(* CODESYS project tctwinsafe.library
   Title: Tc2_TwinSAFE
   Version: 1.0.0.0
   Placeholder: Tc2_TwinSAFE
   Company: Beckhoff Automation GmbH

Project tree, tasks and I/O mapping:
  libraries: Tc2_System, * (Beckhoff Automation GmbH)
  Data types/
    data type TwinSAFE_Data
  Global Variables/
    global variables Globale_Variablen
  POUs/
    function F_GetVersionTcTwinSAFE [ST]
    function block FB_TwinSAFE_connection [ST]
  Version/
    global variables Global_Version
  Visualizations/
*)

// Data types/TwinSAFE_Data
TYPE TwinSAFE_Data :
ARRAY[0..5] OF BYTE;
END_TYPE

// Global Variables/Globale_Variablen
VAR_GLOBAL
END_VAR

// Version/Global_Version
// This function has been automatically generated from the project information.
VAR_GLOBAL CONSTANT
	{attribute 'const_non_replaced'}
	stLibVersion_Tc2_TwinSAFE : ST_LibVersion := (iMajor := 1, iMinor := 0, iBuild := 0, iRevision := 0, sVersion := '1.0.0.0');
END_VAR

// POUs/F_GetVersionTcTwinSAFE
(*
DATE          | Version    | created under        | Author          | Remark
----------------------------------------------------------------------------------------
01/09/2008    | 0.0.1      | V2.10.0 (Build 1321) | O. Ellerbrock   | start of implementation
02/28/2008    | 1.0.0      | V2.10.0 (Build 1323) | O. Ellerbrock   | Release
*)
FUNCTION F_GetVersionTcTwinSAFE : UINT
VAR_INPUT
       nVersionElement       :       INT;
END_VAR
VAR
END_VAR


CASE nVersionElement OF
1: (* major number *)
       F_GetVersionTcTwinSAFE := 1;
2: (* minor number *)
       F_GetVersionTcTwinSAFE := 0;
3: (* revision number *)
       F_GetVersionTcTwinSAFE := 0;
ELSE
   F_GetVersionTcTwinSAFE := 16#FFFF;
END_CASE

END_FUNCTION

// POUs/FB_TwinSAFE_connection
FUNCTION_BLOCK FB_TwinSAFE_connection
(*
The function block FB_TwinSAFE_connection is made for evaluating the TwinSAFE data which is transfered 
from one TwinSAFE communication partner to another TwinSAFE communication partner. The input 
parameters has to be linked to the SafetyQBx or SafetyIn signal of the corresponding TwinSAFE terminal. 
Please assure that the new linkage does not remove the already existing linkage. When RT Ethernet is used 
to transfer the TwinSAFE data, one parameter has to be linked to SafetyQBx the other parameter has to be linked 
to Vardata of the network variable subscriber. 
*)
VAR_INPUT
	TwinSAFETerminal AT %I* : TwinSAFE_Data; (* Additional link to "SafetyIn" e.g. KL1904, KL2904, network variable subscriber*)
	TwinSAFELogic AT %I* : TwinSAFE_Data; (* Additional link to "SafetyQBx" e.g. KL6904 *)
END_VAR
VAR_OUTPUT
	nSafeTerminalData : BYTE; (* TwinSAFE data of SafetyIn e.g. KL1904, KL2904, network variable subscriber *)
	nSafeLogicData : BYTE; (* TwinSAFE data of SafetyOut *)
	tCycleTime: TIME; (* Cycletime in ms *)
	bConnectionInRun : BOOL; (* Connection in RUN *)
	nFirstError : WORD; (* First error in connection *)
	nLastError : WORD; (* Last error in connection *)
END_VAR


VAR
	TwinSAFE_OldInMessage : TwinSAFE_Data;
	OldInCounter : UDINT;
	bConnectionInInRun : BOOL;
	bConnectionOutInRun : BOOL;
	nErrorIn1 : BYTE;
	nErrorIn11 : BYTE;
	nErrorIn2 : BYTE;
	nErrorOut1 : BYTE;
	nErrorOut11 : BYTE;
	nErrorOut2 : BYTE;
	nLastErrorTemp : WORD; (* Last error in connection *)
	Tasknummer: INT := 1; (* Tasknumber of task in which this FB is executed *)
	GETCURTASKINDEX_1: GETCURTASKINDEX;
END_VAR

(* Get Tasknumber of task in which this FB is executed *)
GETCURTASKINDEX_1();
Tasknummer := GETCURTASKINDEX_1.index;

(* Input TwinSAFETerminal *)
CASE TwinSAFETerminal[0] OF

0: (* TwinSAFE *)
	IF TwinSAFETerminal[2] = 0 AND NOT
		(TwinSAFETerminal[1] = 0 AND TwinSAFETerminal[3] = 0 AND TwinSAFETerminal[4] = 0 AND TwinSAFETerminal[5] = 0) THEN
		nSafeTerminalData := TwinSAFETerminal[1];
		bConnectionInInRun := TRUE;
	ELSE
		nSafeTerminalData := 0;
		bConnectionInInRun := FALSE;
	END_IF
	(* Checking for errors *)
	IF TwinSAFETerminal[2] <> 0 AND NOT
		(TwinSAFETerminal[4] = 0 AND TwinSAFETerminal[5] = 0) THEN
		nErrorIn1 := TwinSAFETerminal[2];
		nErrorIn11 := TwinSAFETerminal[0];
	END_IF

	(* Zeitmessung *)
	IF TwinSAFETerminal[3] <> TwinSAFE_OldInMessage[3] THEN
		tCycleTime := UDINT_TO_TIME(((TwinCAT_SystemInfoVarList._TaskInfo[Tasknummer].CycleCount -
		OldInCounter)*  TwinCAT_SystemInfoVarList._TaskInfo[Tasknummer].CycleTime)/10000);
		IF OldInCounter = 0 THEN
			tCycleTime := t#0ms;
		END_IF
		OldInCounter :=  TwinCAT_SystemInfoVarList._TaskInfo[Tasknummer].CycleCount;
		TwinSAFE_OldInMessage := TwinSAFETerminal;
	END_IF

1: (* TwinSAFE *)
	IF TwinSAFETerminal[2] = 0 AND NOT
		(TwinSAFETerminal[4] = 0 AND TwinSAFETerminal[5] = 0) THEN
		nSafeTerminalData := TwinSAFETerminal[1];
		bConnectionInInRun := TRUE;
	ELSE
		nSafeTerminalData := 0;
		bConnectionInInRun := FALSE;
	END_IF
	(* Checking for errors *)
	IF TwinSAFETerminal[2] <> 0 AND NOT
		(TwinSAFETerminal[4] = 0 AND TwinSAFETerminal[5] = 0) THEN
		nErrorIn1 := TwinSAFETerminal[2];
		nErrorIn11 := TwinSAFETerminal[0];
	END_IF

	(* Zeitmessung *)
	IF TwinSAFETerminal[3] <> TwinSAFE_OldInMessage[3] THEN
		tCycleTime := UDINT_TO_TIME(((TwinCAT_SystemInfoVarList._TaskInfo[Tasknummer].CycleCount -
		OldInCounter)*  TwinCAT_SystemInfoVarList._TaskInfo[Tasknummer].CycleTime)/10000);
		IF OldInCounter = 0 THEN
			tCycleTime := t#0ms;
		END_IF
		OldInCounter :=  TwinCAT_SystemInfoVarList._TaskInfo[Tasknummer].CycleCount;
		TwinSAFE_OldInMessage := TwinSAFETerminal;
	END_IF


16#08, 16#2A, 16#4E, 16#52, 16#64: (* Safety over EtherCAT, FailSafe-Data *)
	nSafeTerminalData := 0;
	bConnectionInInRun := FALSE;
	(* Checking for error *)
	IF TwinSAFETerminal[0] = 16#2A THEN
		nErrorIn2 := TwinSAFETerminal[1];
	END_IF
	(* Zeitmessung *)
	IF (TwinSAFETerminal[2] <> TwinSAFE_OldInMessage[2]) OR
		(TwinSAFETerminal[3] <> TwinSAFE_OldInMessage[3])  THEN
		tCycleTime := UDINT_TO_TIME(((TwinCAT_SystemInfoVarList._TaskInfo[Tasknummer].CycleCount -
		OldInCounter)*  TwinCAT_SystemInfoVarList._TaskInfo[Tasknummer].CycleTime)/10000);
		IF OldInCounter = 0 THEN
			tCycleTime := t#0ms;
		END_IF
		OldInCounter :=  TwinCAT_SystemInfoVarList._TaskInfo[Tasknummer].CycleCount;
		TwinSAFE_OldInMessage := TwinSAFETerminal;
	END_IF

16#36: (* Safety over EtherCAT, Data*)
	nSafeTerminalData := TwinSAFETerminal[1];
	bConnectionInInRun := TRUE;
	(* Zeitmessung *)
	IF (TwinSAFETerminal[2] <> TwinSAFE_OldInMessage[2]) OR
		(TwinSAFETerminal[3] <> TwinSAFE_OldInMessage[3])  THEN
		tCycleTime := UDINT_TO_TIME(((TwinCAT_SystemInfoVarList._TaskInfo[Tasknummer].CycleCount -
		OldInCounter)*  TwinCAT_SystemInfoVarList._TaskInfo[Tasknummer].CycleTime)/10000);
		IF OldInCounter = 0 THEN
			tCycleTime := t#0ms;
		END_IF
		OldInCounter :=  TwinCAT_SystemInfoVarList._TaskInfo[Tasknummer].CycleCount;
		TwinSAFE_OldInMessage := TwinSAFETerminal;
	END_IF

ELSE
(* Inputs auf 0 setzen *)
	nSafeTerminalData := 0;
	tCycleTime := t#0ms;
	bConnectionInInRun := FALSE;
END_CASE



(* Input TwinSAFELogic *)
CASE TwinSAFELogic[0] OF

0: (* TwinSAFE Protokoll *)
	IF TwinSAFELogic[2] = 0 AND NOT
		(TwinSAFELogic[4] = 0 AND TwinSAFELogic[5] = 0) THEN
		nSafeLogicData := TwinSAFELogic[1];
		bConnectionOutInRun := TRUE;
	ELSE
		nSafeLogicData := 0;
		bConnectionOutInRun := FALSE;
	END_IF
	(* Checking for errors *)
	IF TwinSAFELogic[2] <> 0 AND NOT
		(TwinSAFELogic[4] = 0 AND TwinSAFELogic[5] = 0) THEN
		nErrorOut1 := TwinSAFELogic[2];
		nErrorOut11 := TwinSAFELogic[0];
	END_IF
1: (* TwinSAFE Protokoll *)
	IF TwinSAFELogic[2] = 0 AND NOT
		(TwinSAFELogic[4] = 0 AND TwinSAFELogic[5] = 0) THEN
		nSafeLogicData := TwinSAFELogic[1];
		bConnectionOutInRun := TRUE;
	ELSE
		nSafeLogicData := 0;
		bConnectionOutInRun := FALSE;
	END_IF
	(* Checking for errors *)
	IF TwinSAFELogic[2] <> 0 AND NOT
		(TwinSAFELogic[4] = 0 AND TwinSAFELogic[5] = 0) THEN
		nErrorOut1 := TwinSAFELogic[2];
		nErrorOut11 := TwinSAFELogic[0];
	END_IF

16#08, 16#2A, 16#4E, 16#52, 16#64: (* Safety over EtherCAT, Failsafe data *)
	nSafeLogicData := 0;
	bConnectionOutInRun := FALSE;
	(* Checking for error *)
	IF TwinSAFELogic[0] = 16#2A THEN
		nErrorOut2 := TwinSAFELogic[1];
	END_IF

16#36: (* Safety over EtherCAT, Process-Data *)
	nSafeLogicData := TwinSAFELogic[1];
	bConnectionOutInRun := TRUE;

ELSE
(* Inputs auf 0 setzen *)
	nSafeLogicData := 0;
	tCycleTime := t#0ms;
	bConnectionOutInRun := FALSE;
END_CASE

(* Setting connection in Run *)
bConnectionInRun := bConnectionInInRun AND bConnectionOutInRun;

(* Resetting the error *)
IF bConnectionInRun THEN
	nFirstError := 0;
	nLastError := 0;
END_IF


(* Setting Firsterror *)
(* Error values
	16#0001: Watchdog in TwinSAFETerminal
	16#0002: Watchdog in TwinSAFELogic
	16#0004: CRC error in TwinSAFETerminal
	16#0008: CRC error in TwinSAFELogic
	16#0010: Slave error in TwinSAFETerminal
	16#0020: Slave error in TwinSAFELogic
	16#4000: not specified error in TwinSAFETerminal
	16#8000: not specified error in TwinSAFELogic
*)
(* Checking where the error occurs first *)
IF nFirstError = 0 THEN (* only for first error executed *)
	(* TwinSAFETerminal *)
	IF nErrorIn1 <> 0 OR nErrorIn2 <> 0 THEN
		IF nErrorIn1 = 16#14 OR nErrorIn2 = 16#04 THEN
			nFirstError := 16#0004;
		ELSIF nErrorIn1 = 16#18 OR nErrorIn2 = 16#05 THEN
			nFirstError := 16#0001;
		ELSIF (nErrorIn1 = 16#10 AND nErrorIn11 = 16#01) OR nErrorIn2 = 16#10 THEN
			nFirstError := 16#0010;
		ELSE
			nFirstError := 16#4000;
		END_IF
	END_IF

	(* TwinSAFELogic *)
	IF nErrorOut1 <> 0 OR nErrorOut2 <> 0 THEN
		IF nErrorOut1 = 16#14 OR nErrorOut2 = 16#04 THEN
			nFirstError := nFirstError OR 16#0008;
		ELSIF nErrorOut1 = 16#18 OR nErrorOut2 = 16#05 THEN
			nFirstError := nFirstError OR 16#0002;
		ELSIF (nErrorOut1 = 16#10 AND nErrorOut11 = 16#01)  OR nErrorOut2 = 16#10 THEN
			nFirstError := nFirstError OR 16#0020;
		ELSE
			nFirstError := nFirstError OR 16#8000;
		END_IF
	END_IF
END_IF

(* Last Error *)
nLastErrorTemp := 0;
(* TwinSAFETerminal *)
IF nErrorIn1 <> 0 OR nErrorIn2 <> 0 THEN
	IF nErrorIn1 = 16#14 OR nErrorIn2 = 16#04 THEN
		nLastErrorTemp := 16#0004;
	ELSIF nErrorIn1 = 16#18 OR nErrorIn2 = 16#05 THEN
		nLastErrorTemp := 16#0001;
	ELSIF (nErrorIn1 = 16#10 AND nErrorIn11 = 16#01) OR nErrorIn2 = 16#10 THEN
		nLastErrorTemp := 16#0010;
	ELSE
		nLastErrorTemp := 16#4000;
	END_IF
END_IF
(* TwinSAFELogic *)
IF nErrorOut1 <> 0 OR nErrorOut2 <> 0 THEN
	IF nErrorOut1 = 16#14 OR nErrorOut2 = 16#04 THEN
		nLastErrorTemp := nLastErrorTemp OR 16#0008;
	ELSIF nErrorOut1 = 16#18 OR nErrorOut2 = 16#05 THEN
		nLastErrorTemp := nLastErrorTemp OR 16#0002;
	ELSIF (nErrorOut1 = 16#10 AND nErrorOut11 = 16#01) OR nErrorOut2 = 16#10 THEN
		nLastErrorTemp := nLastErrorTemp OR 16#0020;
	ELSE
		nLastErrorTemp := nLastErrorTemp OR 16#8000;
	END_IF
END_IF

IF nLastErrorTemp <> nLastError THEN
	nLastError := nLastErrorTemp;
END_IF

(* Reset internal error values *)
nErrorIn1 := 0;
nErrorOut1 := 0;
nErrorIn2 := 0;
nErrorOut2 := 0;

END_FUNCTION_BLOCK
